(* PLC project dc_motor2023_1, Dassault Systèmes ControlBuild 2024x Refresh1 *)
(* stored: creationDateTime 2024-03-18T11:53:50-01:00 *)

FUNCTION_BLOCK stimuli_model
  VAR_OUTPUT
    M_load : REAL := 0.0;
    U : REAL := 0.0;
  END_VAR


ACTION C_source_code:

END_ACTION
END_FUNCTION_BLOCK

FUNCTION_BLOCK edrive_mass_spec
  VAR_INPUT
    M_A : REAL := 0.0;
    M_B : REAL := 0.0;
  END_VAR
  VAR_OUTPUT
    wA : REAL := 0.0;
    phiB : REAL := 0.0;
    phiA : REAL := 0.0;
    wB : REAL := 0.0;
  END_VAR


ACTION C_source_code:

END_ACTION
END_FUNCTION_BLOCK

FUNCTION_BLOCK emachine_model
  VAR_INPUT
    phi : REAL := 0.0;
    U : REAL := 0.0;
    w : REAL := 0.0;
  END_VAR
  VAR_OUTPUT
    I : REAL := 0.0;
    M : REAL := 0.0;
  END_VAR


ACTION C_source_code:

END_ACTION
END_FUNCTION_BLOCK

PROGRAM sut
  VAR_INPUT
    M_load : REAL := 0.0;
    U : REAL := 0.0;
  END_VAR
  VAR_OUTPUT
    phiB : REAL := 0.0;
    M_mot : REAL := 0.0;
    I : REAL := 0.0;
    wB : REAL := 0.0;
  END_VAR

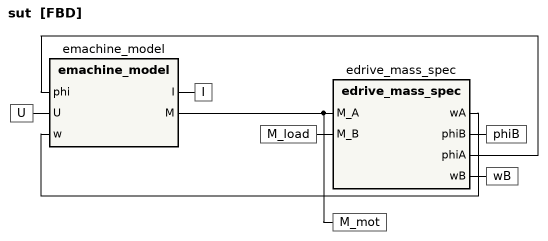
(* FBD diagram, written out as Structured Text *)
emachine_model(phi := edrive_mass_spec.phiA, U := U, w := edrive_mass_spec.wA);
edrive_mass_spec(M_A := emachine_model.M, M_B := M_load);
phiB := edrive_mass_spec.phiB;
M_mot := emachine_model.M;
I := emachine_model.I;
wB := edrive_mass_spec.wB;
END_PROGRAM

PROGRAM dc_motor
  VAR_OUTPUT
    M_mot : REAL := 0.0;
    wB : REAL := 0.0;
    U : REAL := 0.0;
    I : REAL := 0.0;
  END_VAR

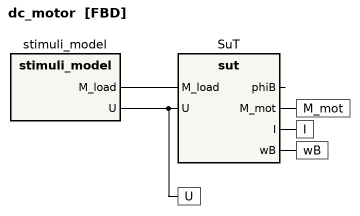
(* FBD diagram, written out as Structured Text *)
stimuli_model();
SuT(M_load := stimuli_model.M_load, U := stimuli_model.U);
M_mot := SuT.M_mot;
wB := SuT.wB;
U := stimuli_model.U;
I := SuT.I;
END_PROGRAM

FUNCTION_BLOCK edrive_mass
  VAR_INPUT
    M_A : REAL := 0.0;
    M_B : REAL := 0.0;
  END_VAR
  VAR_OUTPUT
    wA : REAL := 0.0;
    wB : REAL := 0.0;
    phiB : REAL := 0.0;
    phiA : REAL := 0.0;
  END_VAR


ACTION C_source_code:

END_ACTION
END_FUNCTION_BLOCK

PROGRAM dc_motor_mechanic
  VAR_OUTPUT
    M : REAL := 0.0;
    wB : REAL := 0.0;
  END_VAR

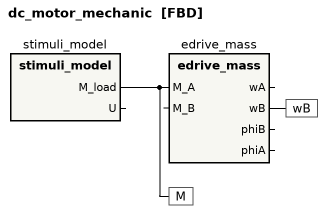
(* FBD diagram, written out as Structured Text *)
stimuli_model();
M := stimuli_model.M_load;
edrive_mass(M_A := stimuli_model.M_load);
wB := edrive_mass.wB;
END_PROGRAM

PROGRAM design_specification_dc_motor_model
  VAR_OUTPUT
    I : REAL := 0.0;
    U : REAL := 0.0;
    M_mot : REAL := 0.0;
    wB : REAL := 0.0;
  END_VAR

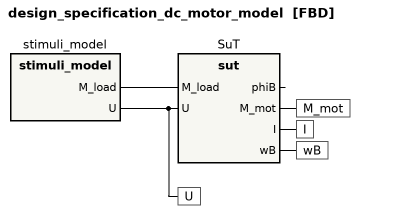
(* FBD diagram, written out as Structured Text *)
stimuli_model();
SuT(M_load := stimuli_model.M_load, U := stimuli_model.U);
I := SuT.I;
U := stimuli_model.U;
M_mot := SuT.M_mot;
wB := SuT.wB;
END_PROGRAM

PROGRAM my_app.dc_motor2023_1

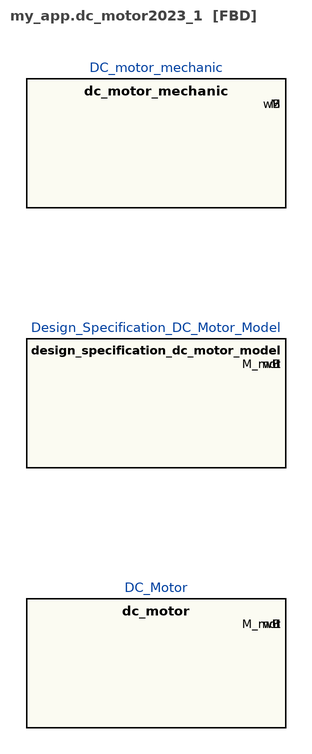
(* FBD diagram, written out as Structured Text *)
DC_motor_mechanic();
Design_Specification_DC_Motor_Model();
DC_Motor();
END_PROGRAM
